// TIA Portal V20 export
DATA_BLOCK "BK04"   // DB308
// stored: MemoryReserve 100
   VAR
      "X10-1.CATHODE MAIN P&P1 LIMITS SENSOR(-)" : Bool := TRUE;
      "X11-1.CATHODE MAIN P&P1 LIMITS SENSOR(+)" : Bool := TRUE;
      "X12-1.CATHODE MAIN P&P2 LIMITS SENSOR(-)" : Bool := TRUE;
      "X13-1.CATHODE MAIN P&P2 LIMITS SENSOR(+)" : Bool := TRUE;
      "X14-1.ANODE MAIN P&P2 LIMITS SENSOR(-)" : Bool := TRUE;
      "X15-1.ANODE MAIN P&P2 LIMITS SENSOR(+)" : Bool := TRUE;
      "X16-1.ANODE MAIN P&P1 LIMITS SENSOR(-)" : Bool := TRUE;
      "X17-1.ANODE MAIN P&P1 LIMITS SENSOR(+)" : Bool := TRUE;
      "X10-2.CATHODE MAIN P&P1 LIMITS SENSOR HOME" : Bool := TRUE;
      "X11-2.SPARE" : Bool := FALSE;
      "X12-2.CATHODE MAIN P&P2 LIMITS SENSOR HOME" : Bool := TRUE;
      "X13-2.SPARE" : Bool := FALSE;
      "X14-2.ANODE MAIN P&P2 LIMITS SENSOR HOME" : Bool := TRUE;
      "X15-2.SPARE" : Bool := FALSE;
      "X16-2.ANODE MAIN P&P1 LIMITS SENSOR HOME" : Bool := TRUE;
      "X17-2.SPARE" : Bool := FALSE;
   END_VAR
BEGIN
END_DATA_BLOCK
